(* PLC project jumps, plcc plcc tests 1 *)
(* stored: creationDateTime 2026-09-27T00:00:00 *)

PROGRAM Jumps
  VAR
    Skip : BOOL;
    Count : INT;
    Always : BOOL;
    Loops : INT;
    Limit : INT := 5;
    Quit : BOOL;
    AfterReturn : BOOL;
  END_VAR

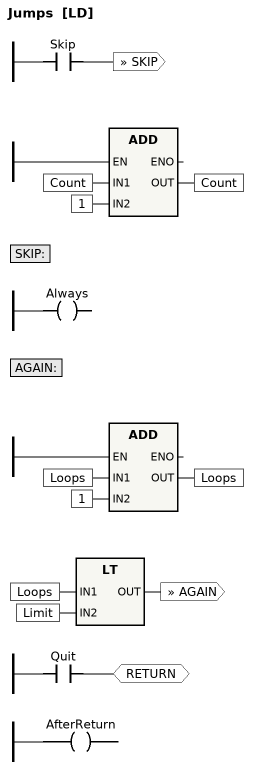
(* LD diagram, written out as Structured Text *)
IF Skip THEN JMP SKIP; END_IF;
Count := Count + 1;
SKIP:
Always := TRUE;
AGAIN:
Loops := Loops + 1;
IF Loops < Limit THEN JMP AGAIN; END_IF;
IF Quit THEN RETURN; END_IF;
AfterReturn := TRUE;
END_PROGRAM
